// TwinCAT 3 PLC project RestApiPlayground
// ProgramVersion: 3.1.4023.0
// libraries:
//   Tc2_Standard, * (Beckhoff Automation GmbH)
//   Tc2_System, * (Beckhoff Automation GmbH)
//   Tc2_Utilities, * (Beckhoff Automation GmbH)
//   Tc3_IotBase, * (Beckhoff Automation GmbH)
//   Tc3_JsonXml, * (Beckhoff Automation GmbH)
//   Tc3_Module, * (Beckhoff Automation GmbH)
// project tree:
//   Abstract/ AwaitableError.TcPOU
//   Blocks/AwaitableErrors/ OnJsonError.TcPOU, OnRequestError.TcPOU
//   Blocks/Callbacks/ FindJsonMember.TcPOU, GetJsonString.TcPOU, IsJsonMemberString.TcPOU, StepChainResetter.TcPOU
//   Blocks/Chains/ TestAwaitChainFast.TcPOU, TestAwaitChainNormal.TcPOU, TestPostLogChain.TcPOU
//   Blocks/ Json.TcPOU, LogBuffer.TcPOU, Await.TcPOU
//   Interfaces/ Awaitable.TcIO, Callable.TcIO, Callback.TcIO, Evaluable.TcIO, Resettable.TcIO
//   / PlcTask.TcTTO
//   Programs/ MAIN.TcPOU
// real-time tasks:
//   TASK PlcTask: cycle T#10ms, priority 20, ADS port 350

CONFIGURATION RestApiPlayground
    RESOURCE PLC ON TwinCAT3
        TASK PlcTask(INTERVAL := T#10ms, PRIORITY := 20);
        PROGRAM MAIN WITH PlcTask : MAIN;
    END_RESOURCE
END_CONFIGURATION

// ---- Interfaces/Awaitable.TcIO
INTERFACE Awaitable EXTENDS Callable, Resettable, Evaluable

METHOD catchIf : Awaitable
VAR_INPUT
	error: BOOL;
	callback: REFERENCE TO AwaitableError;
	message: STRING(255);
END_VAR
END_METHOD

METHOD continueIf : Awaitable
VAR_INPUT
	value: BOOL;
END_VAR
END_METHOD

METHOD evalue : Awaitable
VAR_INPUT
	value: BOOL;
	onTrueCallback: Callback;
	onFalseCallback: REFERENCE TO AwaitableError;
	message: STRING(255);
END_VAR
END_METHOD

METHOD raiseIf : Awaitable
VAR_INPUT
	error: BOOL;
	callback: REFERENCE TO AwaitableError;
	message: STRING(255);
END_VAR
END_METHOD

END_INTERFACE

// ---- Interfaces/Callable.TcIO
INTERFACE Callable

METHOD call : Awaitable
VAR_INPUT
	callback: Callback;
END_VAR
END_METHOD

END_INTERFACE

// ---- Interfaces/Callback.TcIO
INTERFACE Callback

// This is method get's exectued by the framework when the callback is triggered.
// It returns a step number which might be used together with Await to jump to a certain chain step
// after the callback code has been executed.
METHOD execute : UDINT
VAR_INPUT
END_VAR
END_METHOD

END_INTERFACE

// ---- Interfaces/Evaluable.TcIO
INTERFACE Evaluable

METHOD evalue : Awaitable
VAR_INPUT
	value: BOOL;
	onTrueCallback: Callback;
	onFalseCallback: REFERENCE TO AwaitableError;
	message: STRING(255);
END_VAR
END_METHOD

END_INTERFACE

// ---- Interfaces/Resettable.TcIO
INTERFACE Resettable

METHOD reset : PVOID
VAR_INPUT
END_VAR
END_METHOD

END_INTERFACE

// ---- Programs/MAIN.TcPOU
PROGRAM MAIN
VAR
	fastChain: TestAwaitChainFast;
	normalChain: TestAwaitChainNormal;
	postChain: TestPostLogChain;
	logBuffer: LogBuffer;
END_VAR

fastChain();
normalChain();
postChain(logBuffer:=logBuffer);

END_PROGRAM

// ---- Blocks/Chains/TestAwaitChainFast.TcPOU
FUNCTION_BLOCK TestAwaitChainFast
VAR
	nState: UDINT := 0;
	await: Await;

	fbClient: FB_IotHttpClient := (
		sHostName:='localhost',
		bKeepAlive:=TRUE,
		tConnectionTimeout:=T#10S,
		nHostPort:=8000
	);
	
	fbRequest: FB_IotHttpRequest;
	sEndpoint: STRING := '/hello-world';
	response: STRING(255);

	fbJson: FB_JsonDomParser;
	
	jsonDoc: SJsonValue;
	jsonMember: SJsonValue;
	isJsonMemberString: BOOL;
	
	RisingEdge: R_TRIG;
	
	bSend: BOOL;
	requestSent: BOOL;
	cycleCounter: INT := 0;
	lenResponse: INT := 0;
	
	// Awaitable Errors
	onRequestError: OnRequestError := (errorName:='Request error', onErrorStep:=500);
	onResponseError: OnRequestError := (errorName:='Response error', onErrorStep:=500);
	onJsonError: OnJsonError := (errorName:='Json error', onErrorStep:=500);
	
	//Callbacks
	findJsonMemberCallback: FindJsonMember := 
	(
		jsonDomParser:=fbJson, 
		jsonReference:=jsonDoc,
		memberReference:=jsonMember
	);
	
	getJsonStringCallback: GetJsonString := 
	(
		jsonDomParser:=fbJson,
		bufferReference:=response,
		memberReference:=jsonMember
	);
	
	isJsonMemberStringCallback: IsJsonMemberString := 
	(
		jsonDomParser:=fbJson,
		memberReference:=jsonMember,
		isStringReference:=isJsonMemberString
	);
	
END_VAR

RisingEdge(CLK:= bSend );
fbClient.Execute();


CASE nState OF
	
	
	000: // Check if client is configured before moving on to the next step
		
		await.continueIf(fbClient.bConfigured);		
	
	
	010: // Waiting for input to start the request process
		
		await.continueIf(RisingEdge.Q);
	
	
	020: // Send the request
	
		cycleCounter := 0;
		
		requestSent := fbRequest.SendRequest(
			sUri:=sEndpoint, 
			fbClient:=fbClient, 
			eRequestType:=ETcIotHttpRequestType.HTTP_Get, 
			0, // payload, 
			0, // payload size  
			0  // header
		);
					
		await.catchIf(fbRequest.bError,onRequestError, 'An error occured while sending the request')
			.continueIf(requestSent);
	
	030: // Check if request was successful
	
		await.catchIf(fbRequest.bError,onRequestError, 'An error occured after sending the request')
			.continueIf(fbRequest.nStatusCode = 200);
			
		cycleCounter := cycleCounter + 1;
	
	040: // Get the Json response 

		jsonDoc := fbRequest.GetJsonDomContent(fbJson);
		findJsonMemberCallback.memberToFind := 'message';
		lenResponse := len(response);
		await.raiseIf(jsonDoc = 0, onJsonError, 'jsonDoc is an invalid pointer')
			.call(findJsonMemberCallback)
			.raiseIf(jsonMember = 0, onJsonError, 'jsonMember is an invalid pointer')
			.call(isJsonMemberStringCallback)
			.raiseIf(NOT isJsonMemberString, onJsonError, 'The type of the message response is not String')
			.call(getJsonStringCallback)
			.evalue(len(response) > 0, 0, onResponseError, 'The length of the response is 0');
					
		
	500: // Error step

			
	
END_CASE

METHOD FB_init : BOOL
VAR_INPUT
	bInitRetains : BOOL; // if TRUE, the retain variables are initialized (warm start / cold start)
	bInCopyCode : BOOL;  // if TRUE, the instance afterwards gets moved into the copy code (online change)
END_VAR
await.setStepPointer := ADR(nState);
await.setIncreaseValue := 10;
END_METHOD

END_FUNCTION_BLOCK

// ---- Blocks/Await.TcPOU
FUNCTION_BLOCK Await IMPLEMENTS Awaitable

VAR_OUTPUT
END_VAR
VAR
	step: POINTER TO UDINT;
	oldStep: UDINT;
	
	errorCatched: BOOL;
	errorRaised: BOOL;
	increaseByValue: UDINT;

	errorCounter: UDINT;
	errorNames : ARRAY [0..cMax] OF STRING;
	errorMessages : ARRAY [0..cMax] OF STRING;
END_VAR
VAR CONSTANT
    cMax    : UDINT := 1000;
END_VAR

METHOD call : Awaitable
VAR_INPUT
	callback: Callback;
END_VAR
call := THIS^;

IF NOT errorRaised
	AND callback <> 0
	THEN
	
	callback.execute();
	
END_IF
END_METHOD

METHOD catchIf : Awaitable
VAR_INPUT
	error: BOOL;
	callback: REFERENCE TO AwaitableError;
	message: STRING(255);
END_VAR
catchIf := THIS^;

IF errorRaised
	THEN
	RETURN;
END_IF

THIS^.errorCatched := THIS^.errorCatched OR error;

IF error
	THEN
	onError(callback, message, 0);
END_IF
END_METHOD

METHOD continueIf : Awaitable
VAR_INPUT
	value: BOOL;
END_VAR
continueIf := THIS^;

// Make sure step is a valid pointer
IF step = 0 
	OR errorRaised
	THEN
	RETURN;
END_IF


IF value AND NOT THIS^.errorCatched
	THEN
	
	step^ := step^ + increaseByValue;

END_IF
END_METHOD

METHOD evalue : Awaitable
VAR_INPUT
	value: BOOL;
	onTrueCallback: Callback;
	onFalseCallback: REFERENCE TO AwaitableError;
	message: STRING(255);
END_VAR
evalue := THIS^;

// Make sure step is a valid pointer
IF step = 0 
	OR errorRaised
	THEN
	RETURN;
END_IF


IF value AND NOT THIS^.errorCatched
	THEN
	
	step^ := step^ + increaseByValue;
	
	IF onTrueCallback <> 0
	THEN
		onTrueCallback.execute();
	END_IF
	
ELSIF NOT value 
	THEN
	onError(onFalseCallback, message, errorCatched);
END_IF
END_METHOD

METHOD PRIVATE onError : PVOID
VAR_INPUT
	callback: REFERENCE TO AwaitableError;
	message: STRING(255);
	errorRef: REFERENCE TO BOOL;
END_VAR
IF __ISVALIDREF(errorRef)
	THEN
	errorRef := TRUE;
END_IF

	
IF __ISVALIDREF(callback)
	THEN
	
	callback.errorMessage := message;
	IF errorCounter <= cMax
		THEN
		errorNames[errorCounter] := callback.getName();
		errorMessages[errorCounter] := callback.getMessage();
		errorCounter := errorCounter + 1;
	END_IF

	oldStep := step^; 
	step^ := callback.execute();
	
END_IF
END_METHOD

METHOD raiseIf : Awaitable
VAR_INPUT
	error: BOOL;
	callback: REFERENCE TO AwaitableError;
	message: STRING(255);
END_VAR
raiseIf := THIS^;

IF errorRaised
	THEN
	RETURN;
END_IF

IF error 
	THEN
	onError(callback, message, errorRaised);
END_IF
END_METHOD

METHOD reset : PVOID
VAR_INPUT
END_VAR

VAR
	i: UDINT;
END_VAR
errorCounter := 0;
FOR i := 0 TO THIS^.cMAX DO
	IF errorNames[i] = ''
		THEN
		EXIT;
	END_IF
    errorNames[i] := '';
	errorMessages[i] := '';
END_FOR 


errorCatched := FALSE;
errorRaised := FALSE;
oldStep := 0;
END_METHOD

PROPERTY setIncreaseValue : UDINT
SET
increaseByValue := setIncreaseValue;
END_SET
END_PROPERTY

PROPERTY PUBLIC setStepPointer : POINTER TO UDINT
SET
step := setStepPointer;
END_SET
END_PROPERTY

END_FUNCTION_BLOCK

// ---- Abstract/AwaitableError.TcPOU
FUNCTION_BLOCK ABSTRACT AwaitableError IMPLEMENTS Callback
VAR_INPUT
	errorName: STRING;
	errorMessage: STRING(255);
	onErrorStep: UDINT := 0;
END_VAR
VAR_OUTPUT
END_VAR
VAR
END_VAR

(* This is method get's exectued by the framework when the callback is triggered.
 It returns a step number which might be used together with Await to jump to a certain chain step
 after the callback code has been executed.*)
METHOD execute : UDINT
execute := onErrorStep;
END_METHOD

METHOD getMessage : String(255)
VAR_INPUT
END_VAR
getMessage := errorMessage;
END_METHOD

METHOD getName : String
VAR_INPUT
END_VAR
getName := errorName;
END_METHOD

END_FUNCTION_BLOCK

// ---- Blocks/Callbacks/IsJsonMemberString.TcPOU
FUNCTION_BLOCK FINAL IsJsonMemberString IMPLEMENTS Callback
VAR_INPUT
	jsonDomParser: REFERENCE TO FB_JsonDomParser;
	memberReference: REFERENCE TO SJsonValue;
	isStringReference: REFERENCE TO BOOL;
END_VAR

(* This is method get's exectued by the framework when the callback is triggered.
 It returns a step number which might be used together with Await to jump to a certain chain step
 after the callback code has been executed.*)
METHOD execute : UDINT
isStringReference := memberReference <> 0 AND_THEN jsonDomParser.IsString(memberReference);
END_METHOD

END_FUNCTION_BLOCK

// ---- Blocks/AwaitableErrors/OnRequestError.TcPOU
FUNCTION_BLOCK FINAL OnRequestError EXTENDS AwaitableError

END_FUNCTION_BLOCK

// ---- Blocks/AwaitableErrors/OnJsonError.TcPOU
FUNCTION_BLOCK FINAL OnJsonError EXTENDS AwaitableError

END_FUNCTION_BLOCK

// ---- Blocks/Json.TcPOU
FUNCTION_BLOCK Json
VAR_INPUT
END_VAR
VAR_OUTPUT
	payload: STRING(255);
END_VAR
VAR
  writer: FB_JsonSaxWriter;
END_VAR

METHOD create : STRING(255)
VAR_INPUT
	fromString: STRING(255);
END_VAR
writer.StartObject();
writer.AddKey('message');
writer.AddString(fromString);
writer.EndObject();
payload := writer.GetDocument();
writer.ResetDocument();
create := payload;
END_METHOD

END_FUNCTION_BLOCK

// ---- Blocks/Callbacks/FindJsonMember.TcPOU
FUNCTION_BLOCK FINAL FindJsonMember IMPLEMENTS Callback
VAR_INPUT
	memberToFind: STRING;
	jsonDomParser: REFERENCE TO FB_JsonDomParser;
	jsonReference: REFERENCE TO SJsonValue;
	memberReference: REFERENCE TO SJsonValue;
END_VAR


(* This is method get's exectued by the framework when the callback is triggered.
 It returns a step number which might be used together with Await to jump to a certain chain step
 after the callback code has been executed.*)
METHOD execute : UDINT
memberReference := jsonDomParser.FindMember(jsonReference, memberToFind);
END_METHOD

END_FUNCTION_BLOCK

// ---- Blocks/Callbacks/GetJsonString.TcPOU
FUNCTION_BLOCK FINAL GetJsonString IMPLEMENTS Callback
VAR_INPUT
	jsonDomParser: REFERENCE TO FB_JsonDomParser;
	bufferReference: REFERENCE TO STRING(255);
	memberReference: REFERENCE TO SJsonValue;
END_VAR


(* This is method get's exectued by the framework when the callback is triggered.
 It returns a step number which might be used together with Await to jump to a certain chain step
 after the callback code has been executed.*)
METHOD execute : UDINT
bufferReference := jsonDomParser.GetString(memberReference);
END_METHOD

END_FUNCTION_BLOCK

// ---- Blocks/Chains/TestAwaitChainNormal.TcPOU
FUNCTION_BLOCK TestAwaitChainNormal
VAR
	nState: UDINT := 0;
	await: Await;

	fbClient: FB_IotHttpClient := (
		sHostName:='localhost',
		bKeepAlive:=TRUE,
		tConnectionTimeout:=T#10S,
		nHostPort:=8000
	);
	
	fbRequest: FB_IotHttpRequest;
	sEndpoint: STRING := '/hello-world';
	response: STRING(255);

	fbJson: FB_JsonDomParser;
	
	jsonDoc: SJsonValue;
	jsonMember: SJsonValue;
	isJsonMemberString: BOOL;
	
	RisingEdge: R_TRIG;
	
	bSend: BOOL;
	requestSent: BOOL;
	cycleCounter: INT := 0;
	lenResponse: INT := 0;
	
	// Awaitable Errors
	onRequestError: OnRequestError := (errorName:='Request error', onErrorStep:=500);
	onResponseError: OnRequestError := (errorName:='Response error', onErrorStep:=500);
	onJsonError: OnJsonError := (errorName:='Json error', onErrorStep:=500);
	
	//Callbacks
	findJsonMemberCallback: FindJsonMember := 
	(
		jsonDomParser:=fbJson, 
		jsonReference:=jsonDoc,
		memberReference:=jsonMember
	);
	
	getJsonStringCallback: GetJsonString := 
	(
		jsonDomParser:=fbJson,
		bufferReference:=response,
		memberReference:=jsonMember
	);
	
	isJsonMemberStringCallback: IsJsonMemberString := 
	(
		jsonDomParser:=fbJson,
		memberReference:=jsonMember,
		isStringReference:=isJsonMemberString
	);
	
END_VAR

RisingEdge(CLK:= bSend );
fbClient.Execute();


CASE nState OF
	
	
	000: // Check if client is configured before moving on to the next step
		
		await.continueIf(fbClient.bConfigured);		
	
	
	010: // Waiting for input to start the request process
		
		await.continueIf(RisingEdge.Q);
	
	
	020: // Send the request
	
		cycleCounter := 0;
		
		requestSent := fbRequest.SendRequest(
			sUri:=sEndpoint, 
			fbClient:=fbClient, 
			eRequestType:=ETcIotHttpRequestType.HTTP_Get, 
			0, // payload, 
			0, // payload size  
			0  // header
		);
					
		await.catchIf(fbRequest.bError,onRequestError, 'An error occured while sending the request')
			.continueIf(requestSent);
	
	030: // Check if request was successful
	
		await.catchIf(fbRequest.bError,onRequestError, 'An error occured after sending the request')
			.continueIf(fbRequest.nStatusCode = 200);
			
		cycleCounter := cycleCounter + 1;
	
	040: // Get JsonDoc and on success call the findJsonMemberCallback

		jsonDoc := fbRequest.GetJsonDomContent(fbJson);
		findJsonMemberCallback.memberToFind := 'message';
		await.evalue(jsonDoc <> 0, findJsonMemberCallback, onJsonError, 'jsonDoc is an invalid pointer');

	050: //	Check if jsonMember is a valid pointer. On success call the isJsonMemberStringCallback
	
		await.evalue(jsonMember <> 0, isJsonMemberStringCallback, onJsonError, 'jsonMember is an invalid pointer');

		
	060: // Check the type of the json response value and on success call the getJsonStringCallback
		
		await.evalue(isJsonMemberString, getJsonStringCallback, onJsonError, 'The type of the message response is not String');
		
	070: // Check the len of the response
	
		await.evalue(len(response) > 0, 0, onResponseError, 'The length of the response is 0');
		
	500: // Error step

			
	
END_CASE

METHOD FB_init : BOOL
VAR_INPUT
	bInitRetains : BOOL; // if TRUE, the retain variables are initialized (warm start / cold start)
	bInCopyCode : BOOL;  // if TRUE, the instance afterwards gets moved into the copy code (online change)
END_VAR
await.setStepPointer := ADR(nState);
await.setIncreaseValue := 10;
END_METHOD

END_FUNCTION_BLOCK

// ---- Blocks/Chains/TestPostLogChain.TcPOU
FUNCTION_BLOCK TestPostLogChain
VAR_IN_OUT
	logBuffer : LogBuffer;
END_VAR
VAR_OUTPUT
END_VAR
VAR
	await: Await;
	step: UDINT; 
	
	client: FB_IotHttpClient := (
		sHostName:='localhost',
		bKeepAlive:=TRUE,
		tConnectionTimeout:=T#10S,
		nHostPort:=8000
	);
	
	request: FB_IotHttpRequest;
	endpoint: STRING := '/log';
	
	fbJson: FB_JsonDomParser;
	jsonDoc: SJsonValue;
	
	json: Json;
	risingEdge: R_TRIG;
	send: BOOL;
	requestOperation: BOOL;
	
	logMessage : STRING(255);

	// Callbacks
	onRequestError : OnRequestError:= (errorName:='TestPostLogChain.OnRequestError', onErrorStep:=500);
	resetStepOnSuccess: StepChainResetter := (stepReference:=step);  
END_VAR
VAR CONSTANT
	cMax : INT := 100;
END_VAR

risingEdge(CLK:=send );
client.Execute();

CASE step OF 
	
	000: // Basic init step
	
		await.continueIf(client.bConfigured AND logBuffer.pop(logMessage));
		
	010:
		
		json.create(logMessage);
		requestOperation := request.SendRequest(
			sUri:= '/log', 
			fbClient:= client, 
			eRequestType:= ETcIotHttpRequestType.HTTP_POST, 
			pContent:= ADR(json.payload), 			
			nContentSize:= len2(ADR(json.payload)), 
			0
		);
		
		await.evalue(requestOperation, resetStepOnSuccess, onRequestError, 'Error during request');

		
END_CASE

METHOD FB_init : BOOL
VAR_INPUT
	bInitRetains : BOOL; // if TRUE, the retain variables are initialized (warm start / cold start)
	bInCopyCode : BOOL;  // if TRUE, the instance afterwards gets moved into the copy code (online change)
END_VAR
await.setStepPointer := ADR(step);
await.setIncreaseValue := 10;
END_METHOD

END_FUNCTION_BLOCK

// ---- Blocks/LogBuffer.TcPOU
FUNCTION_BLOCK LogBuffer
VAR_INPUT
END_VAR
VAR_OUTPUT
END_VAR
VAR
	logMessages : ARRAY [0..cMax] OF STRING(255);
	counter: INT := 0;
END_VAR
VAR CONSTANT
	cMax: INT := 100;
END_VAR

METHOD append : BOOL
VAR_INPUT
	message: STRING(255);
END_VAR
IF counter <= cMax
	THEN
	
	logMessages[counter] := message;
	counter := counter + 1;
	append := TRUE;
ELSE
	append := FALSE;
END_IF
END_METHOD

PROPERTY logAvailable : Bool
GET
logAvailable := (counter > 0);
END_GET
END_PROPERTY

METHOD pop : BOOL
VAR_IN_OUT
	message : STRING(255);
END_VAR
VAR
	popMessage: INT;
END_VAR
IF counter = 0 AND logMessages[counter] = ''
	THEN
	
	pop := FALSE;
	
ELSIF counter > 0
	THEN
	
	pop := TRUE;
	
	popMessage := counter - 1;
	message := logMessages[popMessage];
	logMessages[popMessage] := '';
	counter := popMessage;
	
END_IF
END_METHOD

END_FUNCTION_BLOCK

// ---- Blocks/Callbacks/StepChainResetter.TcPOU
FUNCTION_BLOCK StepChainResetter IMPLEMENTS Callback
VAR_INPUT
	stepReference:REFERENCE TO UDINT;
END_VAR
VAR_OUTPUT
END_VAR
VAR
END_VAR


(* This is method get's exectued by the framework when the callback is triggered.
 It returns a step number which might be used together with Await to jump to a certain chain step
 after the callback code has been executed.*)
METHOD execute : UDINT
stepReference := 0;
END_METHOD

END_FUNCTION_BLOCK
